FUNCTION F_MeanDirection : LREAL
VAR_INPUT
	direction1,
	direction2: LREAL;
END_VAR
VAR
END_VAR

F_MeanDirection := MODABS(direction1 + 360.0 + direction2 + 360, 360.0);

END_FUNCTION

(* stored: Version 1.1.0.1, ProductVersion 3.1.4024.0
   POU F_MeanDirection: Id {94e882ea-c222-451c-8427-c100167c90fa}, SpecialFunc None *)
